(* CODESYS project Testment_Cartesian_Laser_Platform_Test.export

Project tree, tasks and I/O mapping:
  Testment_Cartesian_Laser_Platform_Test/
    program Cartesian_Laser_Circle_Testment [ST]
*)

// Testment_Cartesian_Laser_Platform_Test/Cartesian_Laser_Circle_Testment
PROGRAM Cartesian_Laser_Circle_Testment	// draw circle as quick as possible
VAR
	
	EnableRobot : BOOL;
	
	enb_axis_and_robot : AuxAxis_PowerOn;
	circle_State : INT;
	col_begain : ARRAY [1..6] OF REAL := [0,0,0,0,0,0];
	row_begain : ARRAY [1..6] OF REAL := [0,0,0,0,0,0];
	col_num_total: BYTE := 10;
	row_num_total : BYTE := 10;
END_VAR


enb_axis_and_robot(enable := EnableRobot);

if not enablerobot then
	circle_State := 0;
END_IF
CASE circle_State OF
	0:
		IF enb_axis_and_robot.Done THEN
			circle_State := 10;
		END_IF
	10:
	
END_CASE

END_PROGRAM
